{attribute addProperty BoxType "EL2521--0000"}
{attribute addProperty Id "StatusAT %I*UINT1621Data_InAT %I*UINT1622"}
{attribute addProperty CRC "1080892866"}
{attribute addProperty SizeInBites "32"}
{attribute addProperty SizeInBytes "4"}
TYPE Inputs_406D1DC2 :
STRUCT
	{attribute addProperty Name "Status"}
	Status AT %I* : UINT;
	{attribute addProperty Name "Data_In"}
	Data_In AT %I* : UINT;
END_STRUCT
END_TYPE

(* stored: Version 1.2.0.0, ProductVersion 3.1.4024.9
   DUT Inputs_406D1DC2: Id {44f96cb1-af53-4c9a-9cc9-5e5f29283f98} *)
